//Alias is a nickname given to type declaration
TYPE myEmployees : ARRAY[1..30] OF myPersonType; END_TYPE

(* stored: Version 1.1.0.1, ProductVersion 3.1.4024.11
   DUT myEmployees: Id {586a2543-cfe2-454a-aee0-3a9edfee8db5} *)
